# EPICS substitutions: simiocApp/Db/sensor.substitutions
file "db/sensor.db"
{

pattern
{SYS,	DEV,	   MEAN,     MSYS,     MDEV }
{sim:,  "dev1:curr",  1.5,   sim:,    "mtr1"}
{sim:,  "dev2:curr",  0.5,   sim:,    "mtr2"}
{sim:,  "dev3:curr", -0.5,   sim:,    "mtr3"}
{sim:,  "dev4:curr", -1.5,   sim:,    "mtr4"}
{sim:,  "dev5:curr", -2.5,   sim:,    "mtr5"}
{sim:,  "dev6:curr", -1.0,   sim:,    "mtr6"}

}
